FUNCTION_BLOCK AI_PUBLISH_1 (* Publish a INT from an AI adapter to one or many SUBSCRIBE_1 Blocks, buffered with a D_FF. Contract: garantiert seit v1.1 einen erzwungenen ersten Publish direkt nach INIT (OPC-UA-Knoten existiert sofort, auch ohne vorherige echte Wertaenderung am Adapter) - dieser erste Publish kann aber noch den Default-/Platzhalterwert des internen Latches enthalten statt des tatsaechlichen aktuellen Adapterwerts, bis die erste echte Aenderung eintrifft. Consumer, die auf den exakten Erstwert angewiesen sind, muessen das beruecksichtigen. Verhalten bei QI=FALSE (deaktivierter Publisher) verifiziert (FORTE-Quellcode, core/src/cominfra/commfb.cpp): weder beim INIT (Verbindung wird geschlossen statt geoeffnet) noch beim erzwungenen Erst-Publish (sendData() bricht vor dem Erreichen der Kommunikationsschicht ab) wird tatsaechlich etwas gesendet oder ein Knoten angelegt - das dabei ausgeloeste CNF/QO=FALSE/STATUS=Inhibited ist reine lokale Rueckmeldung, keine Netzwerkoperation, unbedenklich. Ein spaeterer QI-Wechsel FALSE->TRUE ohne erneutes INIT loest den erzwungenen Erst-Publish NICHT erneut aus. *)
  (* Standard: 61499-2; Description: Copyright (c) 2026 HR Agrartechnik GmbH This program and the accompanying materials are made available under the terms of the Eclipse Public License 2.0 which is available at https://www.eclipse.org/legal/epl-2.0/ SPDX-License-Identifier: EPL-2.0 *)
  (* Version 1.1, 2026-09-17, Franz Höpfinger, HR Agrartechnik GmbH, Erzwungener Erst-Publish nach INIT: PUBLISH_1/PUBLISH_2.INITO -> .REQ ergaenzt (Franz, gegen fehlende OPC-UA-Knoten wenn seit Power-On noch keine echte Wertaenderung stattfand, siehe BERICHT_2026-09-16_STG3_I1_I3_I4_I6_STALE_REMOTE_SUBSCRIBE.md Abschnitt 18-20) - garantiert einen unbedingten ersten Publish direkt nach der Initialisierung. *)
  (* Version 1.0, 2026-08-07, Franz Höpfinger, HR Agrartechnik GmbH, initial API and implementation and/or initial documentation *)
  PACKAGE adapter::net;
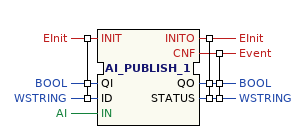
  EVENT_INPUT
    INIT : EInit WITH QI, ID; (* Initialization *)
  END_EVENT
  EVENT_OUTPUT
    INITO : EInit WITH QO, STATUS; (* Initialization Confirm *)
    CNF WITH QO, STATUS; (* Data was sent *)
  END_EVENT
  VAR_INPUT
    QI : BOOL;
    ID : WSTRING;
  END_VAR
  VAR_OUTPUT
    QO : BOOL;
    STATUS : WSTRING;
  END_VAR
  SOCKETS
    IN : adapter::types::unidirectional::AI; (* INT to publish *)
  END_SOCKETS
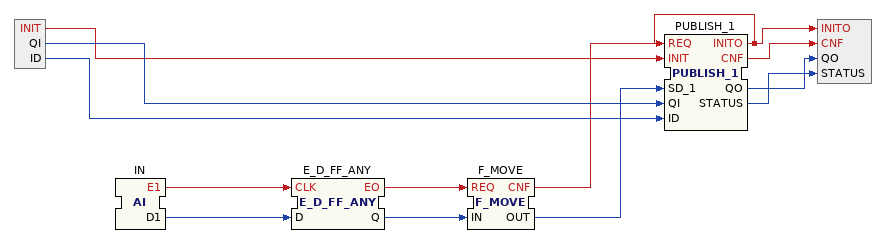
  FBS
    E_D_FF_ANY : iec61499::events::E_D_FF_ANY;
    F_MOVE : iec61131::selection::F_MOVE; {SET_ATTRIBUTE(DataType, INT)}
    PUBLISH_1 : iec61499::net::PUBLISH_1;
  END_FBS
  EVENT_CONNECTIONS
    PUBLISH_1.INITO TO INITO;
    PUBLISH_1.CNF TO CNF;
    IN.E1 TO E_D_FF_ANY.CLK;
    E_D_FF_ANY.EO TO F_MOVE.REQ;
    F_MOVE.CNF TO PUBLISH_1.REQ;
    INIT TO PUBLISH_1.INIT;
    PUBLISH_1.INITO TO PUBLISH_1.REQ;
  END_CONNECTIONS
  DATA_CONNECTIONS
    PUBLISH_1.QO TO QO;
    PUBLISH_1.STATUS TO STATUS;
    IN.D1 TO E_D_FF_ANY.D;
    E_D_FF_ANY.Q TO F_MOVE.IN;
    F_MOVE.OUT TO PUBLISH_1.SD_1;
    QI TO PUBLISH_1.QI;
    ID TO PUBLISH_1.ID;
  END_CONNECTIONS
END_FUNCTION_BLOCK
